// TwinCAT 3 PLC project _16435
// ProgramVersion: 3.1.4023.0
// libraries:
//   Tc2_Standard, * (Beckhoff Automation GmbH)
//   Tc2_System, * (Beckhoff Automation GmbH)
//   Tc3_Module, * (Beckhoff Automation GmbH)
// project tree:
//   GVLs/ INPUT.TcGVL, MOBILEHOIST.TcGVL, OUTPUT.TcGVL
//   / PlcTask.TcTTO
//   POUs/ BLINK.TcPOU, DEADMANCONTROL.TcPOU, ERROR_CASE_STATEMENT.TcPOU, IOSTATE.TcPOU, LIGHTLOGIC.TcPOU, LOADINGLOGIC.TcPOU, MAIN.TcPOU, IO.TcPOU
// real-time tasks:
//   TASK PlcTask: cycle T#10ms, priority 20, ADS port 350
// I/O:
//   DEVICE Device 1 (Beckhoff CCAT)
//   DEVICE Device 2 (EtherCAT), AmsNetId 192.168.128.235.3.1
//     CX8190 [EK1200-5000 EtherCAT Power supply (2A E-Bus)]
//       CX8190 - EL1859 - 1 [EL1859 8Ch. Dig. Input 24V, 3ms, 8Ch. Dig. Output 24V, 0.5A]
//       CX8190 - EL1859 - 2 [EL1859 8Ch. Dig. Input 24V, 3ms, 8Ch. Dig. Output 24V, 0.5A]
//       CX8190 - EL6751 - 1 [EL6751 CANopen Master]
//       Term 5 (EL9011) [EL9011 End Terminal]
//   DEVICE Device 3 (EL6751), AmsNetId 192.168.128.235.4.1
// variable links:
//   16435/16435 Instance <-> Device 2 (EtherCAT)/CX8190/CX8190 - EL1859 - 1
//     PlcTask Inputs/INPUT.EL1859_1 <-> Channel 1/SYSTEM RESET
//     PlcTask Inputs/INPUT.EL1859_1 @bit 1 <-> Channel 2/E-STOP CONDITION
//     PlcTask Inputs/INPUT.EL1859_1 @bit 2 <-> Channel 3/FLOOR POSITION ENABLE SWITCH 1
//     PlcTask Inputs/INPUT.EL1859_1 @bit 3 <-> Channel 4/FLOOR POSITION ENABLE SWITCH 2
//     PlcTask Inputs/INPUT.EL1859_1 @bit 4 <-> Channel 5/THERMOSTAT TEMPERATURE SWITCH
//     PlcTask Inputs/INPUT.EL1859_1 @bit 5 <-> Channel 6/DEADMAN SWITCH
//     PlcTask Inputs/INPUT.EL1859_1 @bit 6 <-> Channel 7/SPARE
//     PlcTask Inputs/INPUT.EL1859_1 @bit 7 <-> Channel 8/SPARE
//     PlcTask Inputs/INPUT.EL1859_1_STATE <-> InfoData/State
//     PlcTask Outputs/OUTPUT.EL1859_1 @bit 1 <-> Channel 10/CONNECTIVITY INDICATOR
//     PlcTask Outputs/OUTPUT.EL1859_1 @bit 2 <-> Channel 11/MAGNETIC BRAKE 1
//     PlcTask Outputs/OUTPUT.EL1859_1 @bit 3 <-> Channel 12/MAGNETIC BRAKE 2
//     PlcTask Outputs/OUTPUT.EL1859_1 @bit 4 <-> Channel 13/INVERTER DC POWER
//     PlcTask Outputs/OUTPUT.EL1859_1 @bit 5 <-> Channel 14/SPOTLIGHT
//     PlcTask Outputs/OUTPUT.EL1859_1 @bit 6 <-> Channel 15/SPARE
//     PlcTask Outputs/OUTPUT.EL1859_1 @bit 7 <-> Channel 16/SPARE
//     PlcTask Outputs/OUTPUT.EL1859_1 <-> Channel 9/SAFETY RELAY RESET SIGNAL
//   16435/16435 Instance <-> Device 2 (EtherCAT)/CX8190/CX8190 - EL1859 - 2
//     PlcTask Inputs/INPUT.EL1859_2 <-> Channel 1/SPARE
//     PlcTask Inputs/INPUT.EL1859_2 @bit {1..7} <-> Channel {2..8}/SPARE  (7 links)
//     PlcTask Inputs/INPUT.EL1859_2_STATE <-> InfoData/State
//     PlcTask Outputs/OUTPUT.EL1859_2 @bit 1 <-> Channel 10/STACK LIGHT AMBER
//     PlcTask Outputs/OUTPUT.EL1859_2 @bit {2..7} <-> Channel {11..16}/SPARE  (6 links)
//     PlcTask Outputs/OUTPUT.EL1859_2 <-> Channel 9/STACK LIGHT RED

CONFIGURATION _16435
    RESOURCE PLC ON TwinCAT3
        TASK PlcTask(INTERVAL := T#10ms, PRIORITY := 20);
        PROGRAM MAIN WITH PlcTask : MAIN;
    END_RESOURCE
END_CONFIGURATION

// ---- GVLs/INPUT.TcGVL
{attribute 'qualified_only'}
VAR_GLOBAL


(*BUS COUPLER 8 INPUTS REFER TO SCHEMATIC CX8190-EL1859-1*)
EL1859_1			AT %I*		:WORD;

(*BUS COUPLER 8 INPUTS REFER TO SCHEMATIC CX8190-EL1859-2*)
EL1859_2			AT %I*		:WORD;

(*BUS COUPLER STATE CX8190-EL1859-1*)
EL1859_1_STATE		AT%I* 		:WORD;

(*BUS COUPLER STATE CX8190-EL1859-2*)
EL1859_2_STATE		AT%I* 		:WORD;

END_VAR

// ---- GVLs/MOBILEHOIST.TcGVL
{attribute 'qualified_only'}
VAR_GLOBAL
	
(*DECLARATION OF INPUTS AND OUTPUTS CORRESPONDING TO MOBILE HOIST.*)


(*INPUTS*)

(*DECLARATION OF RESET SWITCH - INPUT 1 EL1859-1 PIN 1*)
SYSTEM_RESET			:BOOL;

(*DECLARATION OF E-STOP CONDITION PER SAFETY RELAY - INPUT 2 EL1859-1 PIN 2*)
ESTOP_CONDITION			:BOOL;

(*DECLARATION OF FLOOR POSITION ENABLE SWITCH 1 - INPUT 3 EL1859-1 PIN 3*)
FLOORPOSITION_SWITCH1	:BOOL;

(*DECLARATION OF FLOOR POSITION ENABLE SWITCH 2 - INPUT 4 EL1859-1 PIN 4*)
FLOORPOSITION_SWITCH2	:BOOL;

(*DECLARATION OF THERMOSTAT TEMPERATURE SWITCH - INPUT 5 EL1859-1 PIN 5*)
(*THERMOSTAT SET TO DEFAULT 60 DEGREES C*)
TEMP_SWITCH				:BOOL;

(*DECLARATION OF PENDANT DEADMAN SWITCH - INPUT 6 EL1859-1 PIN 6*)
DEADMAN_SWITCH			:BOOL;


(*OUTPUTS*)

(*DECLARATION OF SAFETY RELAY RESET SIGNAL(AMBER) - OUTPUT 1 EL1859-1 PIN 9*)
RESETPB_LED				:BOOL;

(*DECLARATION OF POWER INDICATOR(GREEN) - OUTPUT 2 EL1859-1 PIN 10*)
SELECTORSW_LED			:BOOL;

(*DECLARATION OF MAGNETIC BRAKE 1 - OUTPUT 4 EL1859-1 PIN 11*)
MAGNETIC_BRAKE1			:BOOL;

(*DECLARATION OF MAGNETIC BRAKE 2 - OUTPUT 5 EL1859-1 PIN 12*)
MAGNETIC_BRAKE2			:BOOL;

(*DECLARATION OF INVERTER DC POWER CONTACTOR - OUTPUT 6 EL1859-1 PIN 13*)
MAINPWR					:BOOL;

(*DECLARATION OF SPOTLIGHT - OUTPUT 6 EL1859-7 PIN 14*)
SPOTLIGHT					:BOOL;

(*DECLARATION OF STACK LIGHT RED - EL1859-2 OUTPUT 1 PIN 9*)
REDSTACKLIGHT			:BOOL;

(*DECLARATION OF STACK LIGHT AMBER - EL1859-2 OUTPUT 2 PIN 10*)
AMBERSTACKLIGHT			:BOOL;


(*STATE*)

(*DECLARATION OF IO STATE*)
IOSTATE1				:BOOL;
IOSTATE2				:BOOL;

(*DECLARATION OF IO STATE ERROR*)
IOERROR					:BOOL;

(*DECLARATION OF MAIN STATE*)
MAINSTATE				:INT;


(*DECLATATION OF LOADED STATUS*)
LOWERED_PROPERLY		:BOOL;
LOWERED_IMPROPERLY		:BOOL;
RAISED_PROPERLY			:BOOL;

END_VAR

// ---- GVLs/OUTPUT.TcGVL
{attribute 'qualified_only'}
VAR_GLOBAL
	
(*BUS COUPLER 8 OUTPUTS REFER TO SCHEMATIC CX8190-EL1859-1*)
EL1859_1			AT %Q*		:WORD;

(*BUS COUPLER 8 OUTPUTS REFER TO SCHEMATIC CX8190-EL1859-2*)
EL1859_2			AT %Q*		:WORD;

END_VAR

// ---- POUs/MAIN.TcPOU
PROGRAM MAIN
VAR
END_VAR

(*
 NAME:		16435-MOBILEHOIST
 CREATED:	10/30/2022 
 AUTHOR:	RRODRIGUEZ-HERNANDEZ
 FIRST PROTOTYPE
*)

DEADMANCONTROL();
ERROR_CASE_STATEMENT();
IOSTATE();
LIGHTLOGIC();
LOADINGLOGIC();
IO();

END_PROGRAM

// ---- POUs/DEADMANCONTROL.TcPOU
PROGRAM DEADMANCONTROL
VAR
	
	DEADMANCONTROLCASE	:INT; (*CASE STATEMENT*)
	
END_VAR

CASE DEADMANCONTROLCASE	OF
	
(*NORMAL OPERATION*)

	0:
	
	MOBILEHOIST.MAGNETIC_BRAKE1 	:= FALSE;
	MOBILEHOIST.MAGNETIC_BRAKE2 	:= FALSE;
	MOBILEHOIST.SPOTLIGHT			:= FALSE;
	
	IF	MOBILEHOIST.DEADMAN_SWITCH THEN
		
	DEADMANCONTROLCASE :=1;
		
	END_IF
	
(*DEADMAN SWITCH IS PRESSED*)	
	
	1:
	
	IF MOBILEHOIST.DEADMAN_SWITCH THEN
		
		MOBILEHOIST.MAGNETIC_BRAKE1 	:= TRUE;
		MOBILEHOIST.MAGNETIC_BRAKE2 	:= TRUE;
		MOBILEHOIST.SPOTLIGHT			:= TRUE;
		
	ELSE
		
		MOBILEHOIST.MAGNETIC_BRAKE1 	:= FALSE;
		MOBILEHOIST.MAGNETIC_BRAKE2 	:= FALSE;
		MOBILEHOIST.SPOTLIGHT			:= FALSE;
		DEADMANCONTROLCASE 				:= 0;
		
	END_IF

END_CASE

END_PROGRAM

// ---- POUs/ERROR_CASE_STATEMENT.TcPOU
PROGRAM ERROR_CASE_STATEMENT
VAR
END_VAR

CASE MOBILEHOIST.MAINSTATE OF
	
(*NORMAL OPERATION*)

	0:
		
	IF MOBILEHOIST.LOWERED_PROPERLY THEN
		
		MOBILEHOIST.MAINPWR			:= TRUE;
	
	END_IF


	
	IF MOBILEHOIST.ESTOP_CONDITION OR MOBILEHOIST.IOERROR OR MOBILEHOIST.TEMP_SWITCH = FALSE THEN
		
		MOBILEHOIST.MAINSTATE := 1;
		
	END_IF
	
	IF MOBILEHOIST.LOWERED_IMPROPERLY THEN
		
		MOBILEHOIST.MAINSTATE := 2;
		
	END_IF
	
	IF MOBILEHOIST.RAISED_PROPERLY THEN
		
		MOBILEHOIST.MAINSTATE := 3;
		
	END_IF
	
(*E-STOP/EMERGENCY MODE*)

	1:
	
	MOBILEHOIST.MAGNETIC_BRAKE1 	:= FALSE;
	MOBILEHOIST.MAGNETIC_BRAKE2 	:= FALSE;
	MOBILEHOIST.MAINPWR				:= FALSE;
	
	IF MOBILEHOIST.ESTOP_CONDITION = FALSE AND MOBILEHOIST.IOERROR = FALSE AND MOBILEHOIST.TEMP_SWITCH = FALSE THEN
		
		MOBILEHOIST.MAINSTATE := 0;
		
	END_IF
	
(*IMPROPERLY LOWERED*)

	2:
	
	MOBILEHOIST.MAGNETIC_BRAKE1 	:= FALSE;
	MOBILEHOIST.MAGNETIC_BRAKE2 	:= FALSE;
	MOBILEHOIST.MAINPWR				:= FALSE;

	IF MOBILEHOIST.LOWERED_IMPROPERLY = FALSE THEN
		
		MOBILEHOIST.MAINSTATE := 0;
		
	END_IF
	
(*PROPERLY RAISED*)
	
	3:
	
	MOBILEHOIST.MAGNETIC_BRAKE1 	:= FALSE;
	MOBILEHOIST.MAGNETIC_BRAKE2 	:= FALSE;
	MOBILEHOIST.MAINPWR				:= FALSE;

	IF MOBILEHOIST.RAISED_PROPERLY = FALSE THEN
		
		MOBILEHOIST.MAINSTATE := 0;
		
	END_IF
	
END_CASE

END_PROGRAM

// ---- POUs/IOSTATE.TcPOU
PROGRAM IOSTATE
VAR
END_VAR


(*EL1859-1 & EL1859-2 STATE*)
IF MOBILEHOIST.IOSTATE1 = FALSE OR MOBILEHOIST.IOSTATE2 = FALSE THEN
	
	MOBILEHOIST.IOERROR		:= TRUE;
	
ELSE
	
	MOBILEHOIST.IOERROR		:= FALSE;
	
END_IF

END_PROGRAM

// ---- POUs/LIGHTLOGIC.TcPOU
PROGRAM LIGHTLOGIC
VAR
	
	REDSTACK	:BLINK;
	AMBERSTACK	:BLINK;
	
	LIGHTS		:INT;

END_VAR

(*RESET LED*)
(*RESET LED ON IF ATTACHMENT GOES INTO E-STOP STATE*)

IF MOBILEHOIST.ESTOP_CONDITION THEN
	
	MOBILEHOIST.RESETPB_LED 	:= TRUE;

ELSE

	MOBILEHOIST.RESETPB_LED		:= FALSE;

END_IF

(*RED STACK LIGHT LED*)
(*RED STACK LIGHT LED ON IF ATTACHMENT GOES INTO E-STOP STATE*)
IF MOBILEHOIST.ESTOP_CONDITION THEN
	
	MOBILEHOIST.REDSTACKLIGHT 	:= TRUE;

(*RED STACK LIGHT LED BLINK IF ATTACHMENT LOSE CONNECTIVITY BETWEEN IO CARDS*)
ELSIF MOBILEHOIST.IOERROR THEN
	

	REDSTACK(ENABLE:= TRUE , PERIOD:= T#500MS , Q=> MOBILEHOIST.REDSTACKLIGHT);

ELSE
	
	MOBILEHOIST.REDSTACKLIGHT 	:=FALSE;
	
END_IF

(*AMBER STACK LIGHT LED*)
(*AMBER STACK LIGHT LED ON IF IMPROPERLY LOWERED IN THE GROUND*)
IF MOBILEHOIST.ESTOP_CONDITION = FALSE THEN

IF MOBILEHOIST.LOWERED_IMPROPERLY THEN
	
	MOBILEHOIST.AMBERSTACKLIGHT 	:=TRUE;

ELSE 

	MOBILEHOIST.AMBERSTACKLIGHT	:=FALSE;
	
END_IF

ELSIF MOBILEHOIST.ESTOP_CONDITION THEN
	
	MOBILEHOIST.AMBERSTACKLIGHT := FALSE;	

END_IF

(*GREEN LIGHT*)
(*GREEN SELECTOR SWITCH LIGHT ON IF ATTACHMENT IS OUT OF FAULTS*)
IF MOBILEHOIST.ESTOP_CONDITION = FALSE THEN
	
IF MOBILEHOIST.LOWERED_PROPERLY THEN
	
	MOBILEHOIST.SELECTORSW_LED := TRUE;
	
ELSE
	
	MOBILEHOIST.SELECTORSW_LED := FALSE;
	
END_IF

ELSIF MOBILEHOIST.ESTOP_CONDITION THEN
	
	MOBILEHOIST.SELECTORSW_LED := FALSE;
	
END_IF

(*DEADMAN LIGHT LED*)

IF MOBILEHOIST.ESTOP_CONDITION OR MOBILEHOIST.IOERROR	THEN
	
	MOBILEHOIST.REDSTACKLIGHT 	:= TRUE;

ELSIF MOBILEHOIST.DEADMAN_SWITCH THEN
	

	REDSTACK(ENABLE:= TRUE , PERIOD:= T#500MS , Q=> MOBILEHOIST.REDSTACKLIGHT);
	
	AMBERSTACK(ENABLE:= TRUE , PERIOD:= T#500MS , Q=> MOBILEHOIST.AMBERSTACKLIGHT);
	
END_IF

END_PROGRAM

// ---- POUs/BLINK.TcPOU
FUNCTIon_BLOCK BLINK
VAR_INPUT

	Enable		:	BOOL;	(* Enable Bit to Start Running *)

	Period		:	TIME;	(* Period for Flashing *)

END_VAR


(* === Output Variables === *)
VAR_OUTPUT

	Q		:	BOOL;	(* Flasher Output Bit *)

END_VAR


(* === Local Variables === *)
VAR

	onPeriod	:	Ton;	(* on Period Timer *)

	offPeriod	:	Ton;	(* off Period Timer *)

END_VAR

VAR ConSTANT
END_VAR

(* === Blink Function Block === *)

(*Control of Internal flash bits*)

IF 	Enable = TRUE	THEN

	onPeriod(IN:= NOT offPeriod.Q, PT := Period/2);
	offPeriod(IN:= onPeriod.Q, PT := Period/2);

	Q	:=	NOT onPeriod.Q;

END_IF;

END_FUNCTION_BLOCK

// ---- POUs/LOADINGLOGIC.TcPOU
PROGRAM LOADINGLOGIC
VAR
END_VAR


(*LOGIC TO DEFINE WHETHER THE MOBILE ATTACHMENT IS LOWERED PROPERLY IN THE GROUND*)
IF MOBILEHOIST.FLOORPOSITION_SWITCH1 AND MOBILEHOIST.FLOORPOSITION_SWITCH2 THEN
	
	MOBILEHOIST.LOWERED_PROPERLY 			:= TRUE;
	MOBILEHOIST.LOWERED_IMPROPERLY			:= FALSE;
	MOBILEHOIST.RAISED_PROPERLY				:= FALSE;
	
(*LOGIC TO DEFINE WHETHER THE MOBILE ATTACHMENT IS IMPROPERLY LOWERED*)	
ELSIF (MOBILEHOIST.FLOORPOSITION_SWITCH1 = FALSE AND MOBILEHOIST.FLOORPOSITION_SWITCH2) OR (MOBILEHOIST.FLOORPOSITION_SWITCH1 AND MOBILEHOIST.FLOORPOSITION_SWITCH2 = FALSE) THEN
	
	MOBILEHOIST.LOWERED_PROPERLY 			:= FALSE;
	MOBILEHOIST.LOWERED_IMPROPERLY			:= TRUE;
	MOBILEHOIST.RAISED_PROPERLY				:= FALSE;
	
ELSE
	
(*LOGIC TO DEFINE WHETHER THE MOBILE ATTACHMENT IS RAISED PROPERLY OF THE GROUND*)	
	IF (MOBILEHOIST.FLOORPOSITION_SWITCH1 = FALSE AND MOBILEHOIST.FLOORPOSITION_SWITCH2 = FALSE) THEN
		
	MOBILEHOIST.LOWERED_PROPERLY 			:= FALSE;
	MOBILEHOIST.LOWERED_IMPROPERLY			:= FALSE;
	MOBILEHOIST.RAISED_PROPERLY				:= TRUE;
		
	END_IF

END_IF

END_PROGRAM

// ---- POUs/IO.TcPOU
PROGRAM IO
VAR
END_VAR

(*
 NAME:		16435-MOBILEHOIST
 CREATED:	10/30/2022 
 AUTHOR:	RRODRIGUEZ-HERNANDEZ
 FIRST PROTOTYPE
*)

(*INPUTS - CX8190-EL1859-1*)
MOBILEHOIST.SYSTEM_RESET					:=INPUT.EL1859_1.0;						//INPUT 1
MOBILEHOIST.ESTOP_CONDITION					:=INPUT.EL1859_1.1 = FALSE;				//INPUT 2
MOBILEHOIST.FLOORPOSITION_SWITCH1			:=INPUT.EL1859_1.2;						//INPUT 3
MOBILEHOIST.FLOORPOSITION_SWITCH2			:=INPUT.EL1859_1.3;						//INPUT 4
MOBILEHOIST.TEMP_SWITCH						:=INPUT.EL1859_1.4;						//INPUT 5
MOBILEHOIST.DEADMAN_SWITCH					:=INPUT.EL1859_1.5;						//INPUT 6

(*OUTPUTS - CX8190-EL1859-1*)
OUTPUT.EL1859_1.0 							:=MOBILEHOIST.RESETPB_LED;				//OUTPUT 1			
OUTPUT.EL1859_1.1                           :=MOBILEHOIST.SELECTORSW_LED;			//OUTPUT 2									
OUTPUT.EL1859_1.2                           :=MOBILEHOIST.MAGNETIC_BRAKE1;			//OUTPUT 3
OUTPUT.EL1859_1.3 							:=MOBILEHOIST.MAGNETIC_BRAKE2;			//OUTPUT 4			
OUTPUT.EL1859_1.4                           :=MOBILEHOIST.MAINPWR;					//OUTPUT 5
OUTPUT.EL1859_1.4                           :=MOBILEHOIST.SPOTLIGHT;				//OUTPUT 6

(*OUTPUTS - CX8190-EL1859-2*)
OUTPUT.EL1859_2.0 							:=MOBILEHOIST.REDSTACKLIGHT;			//OUTPUT 1			
OUTPUT.EL1859_2.1                           :=MOBILEHOIST.AMBERSTACKLIGHT;			//OUTPUT 2		

(*STATE*)
MOBILEHOIST.IOSTATE1						:=INPUT.EL1859_1_STATE.3;
MOBILEHOIST.IOSTATE2						:=INPUT.EL1859_2_STATE.3;

END_PROGRAM
